SUBAPPLICATION GBSD_Auswahl (* Waehlt per Button die bodenbasierte Geschwindigkeit/Distanz (GBSD) als Quelle aus, merkt sich die Auswahl persistent im NVS, setzt bei Auswahl die anderen Quellen zurueck und liefert die GBSD-Sensordaten nach aussen *)
  (* Standard: 61499-2 *)
  (* Version 1.0, 2026-08-27, Franz *)
  PACKAGE FBs::Baumsetzer::func::Automatik;
  IMPORT NVS_Keys::Key_GBSD_Store;
  IMPORT isobus::UT::io::Button::ButtonActivationCode::BT_RELEASED_UNLATCHED;
  IMPORT test::FBs::Baumsetzer::Constants::DefaultPool::Button_GBSD;
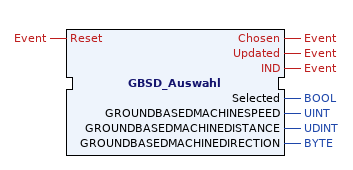
  EVENT_INPUT
    Reset; (* Anforderung von einer der anderen Quellen: eigene Auswahl zuruecksetzen *)
  END_EVENT
  EVENT_OUTPUT
    Chosen; (* Button_GBSD wurde gedrueckt: eigene Auswahl setzen und alle anderen Quellen zuruecksetzen *)
    Updated; (* Ausgewaehlt-Status verfuegbar bzw. geaendert (Init-Lesen oder Aenderung); Trigger fuer nachgelagerte Verarbeitung (u.a. Hintergrundfarbe) *)
    IND; (* Neue GBSD-Daten empfangen (Indication von I_GBSD) *)
  END_EVENT
  VAR_OUTPUT
    Selected : BOOL; (* TRUE wenn GBSD aktuell als Geschwindigkeitsquelle ausgewaehlt ist *)
    GROUNDBASEDMACHINESPEED : UINT; (* Bodenbasierte Maschinengeschwindigkeit (PGN 65097, SPN 1859) *)
    GROUNDBASEDMACHINEDISTANCE : UDINT; (* Bodenbasierte Maschinendistanz (PGN 65097, SPN 1860) *)
    GROUNDBASEDMACHINEDIRECTION : BYTE; (* Bodenbasierte Fahrtrichtung (PGN 65097, SPN 1861) *)
  END_VAR
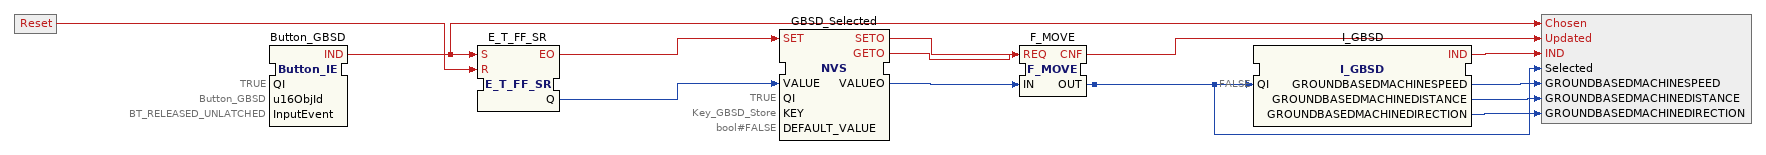
  FBS
    Button_GBSD : isobus::UT::io::Button::Button_IE(QI := TRUE, u16ObjId := Button_GBSD, InputEvent := BT_RELEASED_UNLATCHED);
    E_T_FF_SR : iec61499::events::E_T_FF_SR;
    GBSD_Selected : logiBUS::storage::esp32_nvs::NVS(QI := TRUE, KEY := Key_GBSD_Store, DEFAULT_VALUE := bool#FALSE);
    F_MOVE : iec61131::selection::F_MOVE; {SET_ATTRIBUTE(DataType, BOOL)}
    I_GBSD : isobus::tecu::I_GBSD(QI := FALSE);
  END_FBS
  EVENT_CONNECTIONS
    Button_GBSD.IND TO E_T_FF_SR.S;
    Button_GBSD.IND TO Chosen;
    Reset TO E_T_FF_SR.R;
    E_T_FF_SR.EO TO GBSD_Selected.SET;
    GBSD_Selected.SETO TO F_MOVE.REQ;
    GBSD_Selected.GETO TO F_MOVE.REQ;
    F_MOVE.CNF TO Updated;
    I_GBSD.IND TO IND;
  END_CONNECTIONS
  DATA_CONNECTIONS
    E_T_FF_SR.Q TO GBSD_Selected.VALUE;
    GBSD_Selected.VALUEO TO F_MOVE.IN;
    F_MOVE.OUT TO I_GBSD.QI;
    F_MOVE.OUT TO Selected;
    I_GBSD.GROUNDBASEDMACHINESPEED TO GROUNDBASEDMACHINESPEED;
    I_GBSD.GROUNDBASEDMACHINEDISTANCE TO GROUNDBASEDMACHINEDISTANCE;
    I_GBSD.GROUNDBASEDMACHINEDIRECTION TO GROUNDBASEDMACHINEDIRECTION;
  END_CONNECTIONS
END_SUBAPPLICATION
